// TIA Portal V19 export
DATA_BLOCK "ItemCommand"   // DB10
{ S7_Optimized_Access := 'TRUE' }
AUTHOR : FLA
FAMILY : UHT
VERSION : 1.0
// stored: AutoNumber false, MemoryReserve 0
   VAR RETAIN
      Y0101 : "ItemCommand_UDT";
      Y0103 : "ItemCommand_UDT";
      Y0104 : "ItemCommand_UDT";
      Y0109 : "ItemCommand_UDT";
      Y0111 : "ItemCommand_UDT";
      Y0112 : "ItemCommand_UDT";
      Y0113 : "ItemCommand_UDT";
      Y0114 : "ItemCommand_UDT";
      Y0115 : "ItemCommand_UDT";
      M0139 : "ItemCommand_UDT";
      Y0116 : "ItemCommand_UDT";
      Y0108 : "ItemCommand_UDT";
      Y0117 : "ItemCommand_UDT";
      Y0118 : "ItemCommand_UDT";
      Y0237 : "ItemCommand_UDT";
      Y0238 : "ItemCommand_UDT";
      Y0119 : "ItemCommand_UDT";
      Y0124 : "ItemCommand_UDT";
      Y0135_NOT_USED : "ItemCommand_UDT";
      Y0136_NOT_USED : "ItemCommand_UDT";
      Y0137_NOT_USED : "ItemCommand_UDT";
      Y0143 : "ItemCommand_UDT";
      Y0144_NOT_USED : "ItemCommand_UDT";
      Y0147 : "ItemCommand_UDT";
      Y0148 : "ItemCommand_UDT";
      Y0158 : "ItemCommand_UDT";
      Y0545 : "ItemCommand_UDT";
      PACK1 : "ItemCommand_UDT";
      PACK2 : "ItemCommand_UDT";
      PACK3 : "ItemCommand_UDT";
      PACK4 : "ItemCommand_UDT";
      AlarmLamp : "ItemCommand_UDT";
      AHV_CLOSED : "ItemCommand_UDT";
      AHV_HIGH_LEVEL : "ItemCommand_UDT";
      AHV_READY : "ItemCommand_UDT";
      AHV_SHUT_DOWN : "ItemCommand_UDT";
      AHV_STERILE : "ItemCommand_UDT";
      PROD_AVAILABLE : "ItemCommand_UDT";
      RINSE_READY : "ItemCommand_UDT";
      CAUSTIC_READY : "ItemCommand_UDT";
      ACID_READY : "ItemCommand_UDT";
      CIP_FILLER_ENABLE : "ItemCommand_UDT";
      WATER_PUMP : "ItemCommand_UDT";
      Y0901 : "ItemCommand_UDT";
      Y0902 : "ItemCommand_UDT";
      Y0903 : "ItemCommand_UDT";
      TANK_READY : "ItemCommand_UDT";
      TANK_OPEN : "ItemCommand_UDT";
      Y0904 : "ItemCommand_UDT";
      Y0905 : "ItemCommand_UDT";
      Y0906 : "ItemCommand_UDT";
      Y0907 : "ItemCommand_UDT";
      Y0908 : "ItemCommand_UDT";
      Y0909 : "ItemCommand_UDT";
      Y0910 : "ItemCommand_UDT";
      Y0911 : "ItemCommand_UDT";
      Y0912 : "ItemCommand_UDT";
      Q41_1 : "ItemCommand_UDT";
      CIP_Route : "ItemCommand_UDT";
      SIP_Steam : "ItemCommand_UDT";
      Product_Available : "ItemCommand_UDT";
      Barrier_Sterile : "ItemCommand_UDT";
      Product_Route : "ItemCommand_UDT";
      X0913 : "ItemCommand_UDT";
      V0930 : "ItemCommand_UDT";
      V0931 : "ItemCommand_UDT";
      spare2 : "ItemCommand_UDT";
      V0552 : "ItemCommand_UDT";
      V0934 : "ItemCommand_UDT";
      V0935 : "ItemCommand_UDT";
      V0940 : "ItemCommand_UDT";
      V0941 : "ItemCommand_UDT";
      V0942 : "ItemCommand_UDT";
      V0943 : "ItemCommand_UDT";
      V0944 : "ItemCommand_UDT";
      V0945 : "ItemCommand_UDT";
      M0940 : "ItemCommand_UDT";
      V1021 : "ItemCommand_UDT";
      V1023 : "ItemCommand_UDT";
      V1024 : "ItemCommand_UDT";
      V1025 : "ItemCommand_UDT";
      V1027 : "ItemCommand_UDT";
      V1083 : "ItemCommand_UDT";
      M0941 : "ItemCommand_UDT";
      V0936 : "ItemCommand_UDT";
   END_VAR
BEGIN
END_DATA_BLOCK
